{attribute 'linkalways'} 
{attribute 'no_explicit_call' := 'This FB is a CLASS and must be accessed using methods or properties'}
{attribute 'enable_dynamic_creation'}
FUNCTION_BLOCK Node_F_VN_ContainerAverageVarianceElementwise4 EXTENDS VisionNode
VAR
    ipSrcContainer : _ITcVnContainer;
    aAverage : _TcVnVector4_LREAL;
	aVariance : _TcVnVector4_LREAL;
    hrPrev : _HRESULT(S_OK);
    hresult : _HRESULT(S_OK);
END_VAR

METHOD PUBLIC  Clone : I_Node
VAR
	pNode : POINTER TO Node_F_VN_ContainerAverageVarianceElementwise4;
END_VAR
pNode := __NEW(Node_F_VN_ContainerAverageVarianceElementwise4);
Clone := pNode^;
END_METHOD

METHOD FB_init : BOOL
VAR_INPUT
	bInitRetains : BOOL; // if TRUE, the retain variables are initialized (warm start / cold start)
	bInCopyCode : BOOL;  // if TRUE, the instance afterwards gets moved into the copy code (online change)
END_VAR
AddInput('ipSrcContainer', ipSrcContainer);
AddInput('hrPrev', hrPrev);
AddOutput('aAverage', aAverage);
AddOutput('aVariance', aVariance);
AddOutput('hresult',hresult);
END_METHOD

METHOD PROTECTED OnExecute
hresult.Value := F_VN_ContainerAverageVarianceElementwise4(
    ipSrcContainer := ipSrcContainer.Value,
    aAverage := aAverage.Value,
	aVariance := aVariance.Value,
    hrPrev:= hrPrev.Value);
END_METHOD

METHOD PUBLIC PreExecutionCheck
VAR_INPUT
	Check : I_PreExecutionChecks;
END_VAR
VAR
	isCorrectType : BOOL;
END_VAR
Check.IsTrue(ipSrcContainer.IsValid, 'ipContainer must be a valid container');

isCorrectType := 
    // ---------------------------------------------------------
    // Vector 4 Types (X, Y, Z, W)
    // ---------------------------------------------------------
    ipSrcContainer.IsType(TC_GLOBAL_CONST_LIST.ContainerType_Vector_TcVnVector4_SINT) OR_ELSE
    ipSrcContainer.IsType(TC_GLOBAL_CONST_LIST.ContainerType_Vector_TcVnVector4_USINT) OR_ELSE
    ipSrcContainer.IsType(TC_GLOBAL_CONST_LIST.ContainerType_Vector_TcVnVector4_INT) OR_ELSE
    ipSrcContainer.IsType(TC_GLOBAL_CONST_LIST.ContainerType_Vector_TcVnVector4_UINT) OR_ELSE
    ipSrcContainer.IsType(TC_GLOBAL_CONST_LIST.ContainerType_Vector_TcVnVector4_DINT) OR_ELSE
    ipSrcContainer.IsType(TC_GLOBAL_CONST_LIST.ContainerType_Vector_TcVnVector4_REAL) OR_ELSE
    ipSrcContainer.IsType(TC_GLOBAL_CONST_LIST.ContainerType_Vector_TcVnVector4_LREAL);

Check.IsTrue(isCorrectType, 'ipContainer contains incorrect type for Elementwise4');
END_METHOD

END_FUNCTION_BLOCK

(* stored: Version 1.1.0.1, ProductVersion 3.1.4026.13
   POU Node_F_VN_ContainerAverageVarianceElementwise4: Id {f75d1910-47e9-00ca-0ec1-bb99c061e72c}, SpecialFunc None
   Folder Constructor: Id {9b2ad974-0af1-0c5d-0272-a769bd689da2}
   Method Clone: Id {6feab672-815f-0f91-1ca1-4c07aaeffe3e}
   Method FB_init: Id {216b2176-9384-0e7e-3421-497d4e86114e}
   Method OnExecute: Id {3987419a-db4c-0497-1edd-da7919d0c2c9}
   Method PreExecutionCheck: Id {e44ecaee-02c8-0f8a-2ad7-15beece09cb6} *)
